FUNCTION_BLOCK FT_DERIV (* Calculate derivative over signal 'in' with Factor 'K' *)
  (* Standard: 61499-1 *)
  (* Version 1.1, 2025-12-21, CodingAssistant *)
  PACKAGE OSCAT::Basic::POUs::Engineering::Control;
  IMPORT OSCAT::Basic::POUs::Engineering::measurements::T_PLC_US;
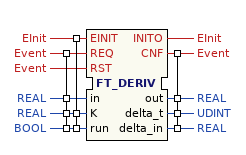
  EVENT_INPUT
    EINIT : EInit WITH K, run; (* Init Request *)
    REQ WITH in, K, run; (* Normal Execution Request *)
    RST; (* Reset *)
  END_EVENT
  EVENT_OUTPUT
    INITO : EInit; (* Init Confirmation *)
    CNF WITH out, delta_t, delta_in; (* Execution Confirmation *)
  END_EVENT
  VAR_INPUT
    in : REAL; (* Input Signal *)
    K : REAL := 1.0; (* Derivation Factor *)
    run : BOOL := 1; (* Enable calculation *)
  END_VAR
  VAR_OUTPUT
    out : REAL; (* Calculated Derivative *)
    delta_t : UDINT; (* Time difference in microseconds *)
    delta_in : REAL; (* Input signal difference *)
  END_VAR
  VAR
    old : REAL;
    tx : UDINT;
    last : UDINT;
    init : BOOL;
  END_VAR
  EC_STATES
    EINIT : EINIT -> INITO;
    REQ : REQ -> CNF;
    RST : RST -> CNF;
  END_STATES
  ALGORITHM EINIT IN ST:
init := FALSE;
  END_ALGORITHM
  ALGORITHM RST IN ST:
init := TRUE;
old := in;
  END_ALGORITHM
  ALGORITHM REQ IN ST:
(* read system time *)
tx := T_PLC_US();
delta_t := tx - last;
last := tx;

(* init on first startup *)
IF NOT init THEN
	this.RST();
ELSIF run AND delta_t > 0 THEN
	delta_in := in - old;
		// Mikrosekunden in Sekunden
	out := delta_in / UDINT_TO_REAL(delta_t) * 1000000.0 * K;
	old := in;
ELSE
	out := 0.0;
END_IF;
  END_ALGORITHM
END_FUNCTION_BLOCK
